TYPE DesignerUserData EXTENDS TcoCore.TcoStruct :
STRUCT
    {attribute addProperty Name "<#ResultBool#>"}
    ResultBool : BOOL;
    {attribute addProperty Name "<#ResultInt#>"}
    ResultInt : INT;
    {attribute addProperty Name "<#ResultString#>"}
    ResultString : STRING;
END_STRUCT
END_TYPE

(* stored: Version 1.1.0.1, ProductVersion 3.1.4024.12
   DUT DesignerUserData: Id {2b54b571-0724-0aed-051f-ae9265f6c6e7} *)
